RoboDK station: ProjetRoboDK_LaBrise.rdk

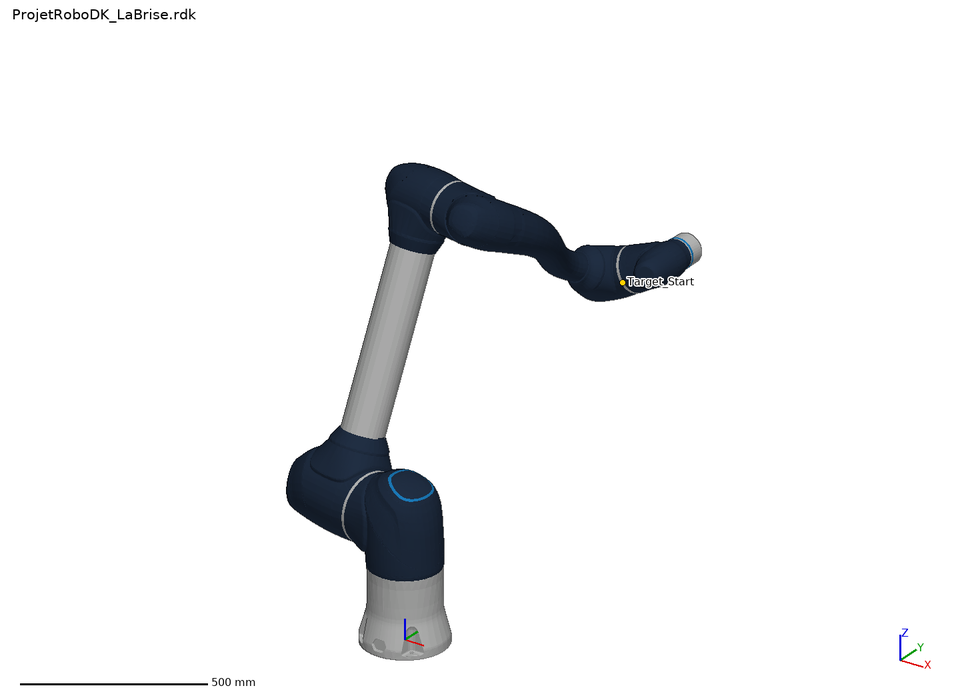
[picture v0: the station drawn from its stored meshes, robots at their saved joint values, targets as dots, program paths as lines]
Station RobotPhoto (saved by RoboDK 5.5.1). Poses are relative to the parent item; angles as X-Y-Z fixed-axis rotations.
  - frame Doosan Robotics H2017 Base at (0, 0, 0) mm
    - robot Doosan Robotics H2017: 6 axes, payload 20 kg, reach 1700 mm, repeatability 0.1 mm
        modified DH rows (alpha deg, a mm, theta deg, d mm): 0, 0, 180, 344.3; -90, 0, -90, -9.9; 0, 845, -90, 0; -90, 0, 0, 734; 90, 0, 0, 0; -90, 0, 180, 121
        joint limits [-360, -130, -160, -360, -360, -360] to [360, 130, 160, 360, 360, 360]; home [0, 0, -90, 0, 0, 0]; saved at [77.365, 20.224, 96.679, -27.985, -29.584, 24.727]
    - target Target_Start (Cartesian target) at (-23.69, 1046.9, 635.51) mm, rotated rx -177.88 ry 89.73 rz -87.12 deg; joints [90.754, 25.463, 104.469, -0.009, -39.662, -0.003] of Doosan Robotics H2017
  - Python program Prog1 (listed below)

--- Python program Prog1 ---
from robodk import robolink    # RoboDK API
from robodk import robomath    # Robot toolbox

from robodk import *      # RoboDK API
from robolink import *    # Robot toolbox

from math import *
from time import sleep

from LaBrise.take_picture import image_viewer

os.system('cls')
cam = image_viewer()

#---[CONNEXION]---#
RDK = Robolink()

robot = RDK.ItemUserPick('Select a robot', ITEM_TYPE_ROBOT)
if not robot.Valid():
    raise Exception('No robot selected or available')

RUN_ON_ROBOT = True

#RDK.setRunMode(RUNMODE_RUN_ROBOT)

if RUN_ON_ROBOT:
    success = robot.Connect()
    status, status_msg = robot.ConnectedState()
    if status != ROBOTCOM_READY:
        print(status_msg)
        raise Exception("Failed to connect: " + status_msg)

    RDK.setRunMode(RUNMODE_RUN_ROBOT)
#-----------------#

def mouvement(LONGUEUR_FOTO, HAUTEUR_FOTO, longueur, hauteur):
    start_pose = RDK.Item('Target_Start').Pose()
    robot.MoveJ(start_pose)

    robot.setPoseFrame(robot.PoseFrame())
    robot.setPoseTool(robot.PoseTool())

    robot.setZoneData(10)
    #robot.setSpeed(50,5)

    #---[CALCUL DU GRID]---#
    num_grid_x = ceil(longueur/LONGUEUR_FOTO)
    overlapping_x = (num_grid_x*LONGUEUR_FOTO - longueur)/(num_grid_x-1)
    grid_x = [(LONGUEUR_FOTO/2)-(longueur/2) + i*(LONGUEUR_FOTO-overlapping_x) for i in range(num_grid_x)]

    num_grid_y = ceil(hauteur/HAUTEUR_FOTO)
    overlapping_y = (num_grid_y*HAUTEUR_FOTO - hauteur)/(num_grid_y-1)
    grid_y = [(HAUTEUR_FOTO/2)-(hauteur/2) + i*(HAUTEUR_FOTO-overlapping_y) for i in range(num_grid_y)]

    grid = []
    for y in range(num_grid_y):
        for x in range(num_grid_x):
            if y%2 == 0:
                grid.append((grid_x[x], grid_y[-y-1]))
            else:
                grid.append((grid_x[-x-1], grid_y[-y-1]))
    #----------------------#

    counter = 1

    target = Mat(start_pose)
    pos = target.Pos()
    pos[2] += grid[0][1]
    pos[0] -= grid[0][0]
    target.setPos(pos)

    robot.MoveJ(target)

    cam.take_picture(sys.argv, str(counter) + '.png')

    sleep(5)
    counter += 1

    for point in grid[1:]:
        target = Mat(start_pose)
        pos = target.Pos()
        pos[2] += point[1]
        pos[0] -= point[0]
        target.setPos(pos)

        robot.MoveJ(target)

        cam.take_picture(sys.argv, str(counter) + '.png')

        sleep(1)
        counter += 1

###
import tkinter as tk
from tkinter import messagebox

### Création de fonctions

def fQuit():
    return app.destroy()

def show_error_window():
    messagebox.showerror("ERREUR", "Veuillez sélectionner des dimmensions non nulles")

def toContinue():
    if(var_entryX.get() == 0 or var_entryY.get() == 0 or var_scaleX.get() == 0 or var_scaleY.get() == 0):
       return show_error_window()
    else :
        '''next_window = tk.Toplevel(app)
        next_window.title("Autre fenetre")
        next_window.geometry("560x480")
        next_window.resizable(False, False)'''

        joints_ref = robot.Joints()

        #print(10*var_entryX,10*var_entryY, 10*var_scaleX, 10*var_scaleY)

        mouvement(var_entryX.get(),var_entryY.get(), var_scaleX.get(), var_scaleY.get())

### Fenetre principale - choix des dimensions

#----------------------------------------------------------------------------------------------------

app = tk.Tk()
app.title("Détection de fissures")
app.geometry("560x480")
app.resizable(False, False)

### Création des variables

var_entryX = tk.IntVar()
var_entryY = tk.IntVar()
var_scaleX = tk.IntVar()
var_scaleY = tk.IntVar()

#----------------------------------------------------------------------------------------------------

frame = tk.LabelFrame(app, text="Taille du mur à scanner(mm)")
scale_x = tk.Scale(frame, from_ = 0, to = 1000, tickinterval = 500, orient="horizontal", length = 200, variable = var_scaleX)
scale_y = tk.Scale(frame, from_ = 0, to = 1000, tickinterval = 500, orient="vertical", length = 200, variable = var_scaleY)

frame2 = tk.LabelFrame(app, text="Taile des images(mm)")
entryX = tk.Entry(frame2, textvariable = var_entryX)
entryY = tk.Entry(frame2, textvariable = var_entryY)
labelX = tk.Label(frame2, text ="X(mm)")
labelY = tk.Label(frame2, text ="Y(mm)")

quit_button = tk.Button(app, text = "Quit", command = fQuit)
continue_button = tk.Button(app, text = "Continue", command = toContinue)


frame.pack(fill = "x")
scale_x.pack()
scale_y.pack(side = "left")


frame2.pack(fill = "x")
entryX.pack()
entryY.pack()
labelX.place(x = 350, y = 0)
labelY.place(x = 350, y = 17)

quit_button.place(x = 10, y = 440)
continue_button.place(x = 480, y = 440)
app.mainloop()
###
